// TwinCAT 3 PLC project PLCSample
// ProgramVersion: 3.1.4024.0
// libraries:
//   Tc2_Standard, * (Beckhoff Automation GmbH)
//   Tc2_System, * (Beckhoff Automation GmbH)
//   Tc3_Module, * (Beckhoff Automation GmbH)
// project tree:
//   DUTs/ FooBar.TcDUT
//   / PlcTask.TcTTO
//   POUs/ MAIN.TcPOU
// real-time tasks:
//   TASK PlcTask: cycle T#10ms, priority 20, ADS port 350

CONFIGURATION PLCSample
    RESOURCE PLC ON TwinCAT3
        TASK PlcTask(INTERVAL := T#10ms, PRIORITY := 20);
        PROGRAM MAIN WITH PlcTask : MAIN;
    END_RESOURCE
END_CONFIGURATION

// ---- DUTs/FooBar.TcDUT
{attribute 'qualified_only'}
{attribute 'strict'}
TYPE FooBar :
(
	FOO_BAR_UNSPECIFIED := 0,
	FOO_BAR_FIRST_VALUE := 1,
	FOO_BAR_SECOND_VALUE := 2
);
END_TYPE

// ---- POUs/MAIN.TcPOU
PROGRAM MAIN
VAR
	bar : FooBar;
END_VAR

bar := FooBar.FOO_BAR_FIRST_VALUE;

END_PROGRAM
